Staubli VAL3: vHome.pgx

program vHome()
  local pointRx l_pHome
  local pointRx l_pLokalnoGor
begin
  nTaskWorking = nTaskWorking + 1
  //l_pHome=jointToPoint(flange,world,jHome)
  cConfigHome=pHome.config
  l_pLokalnoGor=here(flange, world)
  // Vedno premakni za visino 60mm
  // Ni pomembno katero orodje je izbrano saj se premikamo po smereh globalnega sistemu
  // Orodje je pomembno tu le za dolocanje trenutne pozicija, a ni vazno kaj izberemo
  // saj orientacije ne bomo spreminjali, prav tako pa je premik relativen oz. je
  // RAZLIKA v visini ENAKA, ne glede na to katero orodje je izbrano
  l_pLokalnoGor.trsf.z= l_pLokalnoGor.trsf.z + 60
  l_pLokalnoGor={l_pLokalnoGor.trsf,cConfigHome}
  movel(l_pLokalnoGor,flange,mSrednje)
  waitEndMove()
  movel(pHome,flange,mSrednje)
  waitEndMove()
  sDiag="Sem v osnovnem položaju"
  nTaskWorking = nTaskWorking - 1
end
